TYPE Vec8d : ARRAY[1..8] OF LREAL; END_TYPE

(* stored: Version 1.1.0.1, ProductVersion 3.1.4024.12
   DUT Vec8d: Id {40be82d6-42a6-43a6-8f5f-26e54fff4236} *)
